(* PLC project shuttle_control, Dassault Systèmes ControlBuild 2024x *)
(* stored: creationDateTime 2023-10-03T11:13:58-01:00 *)

FUNCTION_BLOCK tri_chain.shuttle_control
  VAR_INPUT
    globalRunning : BOOL := false;
    sensorPos1 : BOOL := false;
    sensorPos2 : BOOL := false;
    sensorPos3 : BOOL := false;
    requestCapture1 : BOOL := false;
    endCapture1 : BOOL := false;
    requestCapture2 : BOOL := false;
    endCapture2 : BOOL := false;
    requestCapture3 : BOOL := false;
    endCapture3 : BOOL := false;
    depositRequest : BOOL := false;
    depositFinished : BOOL := false;
  END_VAR
  VAR_OUTPUT
    enableCapture1 : BOOL := false;
    enableCapture2 : BOOL := false;
    enableCapture3 : BOOL := false;
    enableCapture : BOOL := false;
    enableDeposit : BOOL := false;
    moveToLeft : BOOL := false;
    moveToRight : BOOL := false;
  END_VAR
  VAR
    goTo1 : BOOL := false;
    goTo2 : BOOL := false;
    goTo3 : BOOL := false;
    shuttleInPosition : BOOL := false;
  END_VAR

INITIAL_STEP 10:
  COMPUTE_FUNCTION_BLOCKS(S);
END_STEP
TRANSITION FROM 10 TO 11
  := requestCapture1 AND globalRunning;
END_TRANSITION
TRANSITION FROM 10 TO 13
  := requestCapture2 AND globalRunning;
END_TRANSITION
TRANSITION FROM 10 TO 15
  := requestCapture3 AND globalRunning;
END_TRANSITION
INITIAL_STEP 20:
END_STEP
TRANSITION FROM 20 TO 21
  := goTo2 AND NOT sensorPos2;
END_TRANSITION
TRANSITION FROM 20 TO 22
  := goTo2 AND sensorPos2;
END_TRANSITION
INITIAL_STEP 30:
END_STEP
TRANSITION FROM 30 TO 31
  := goTo1 AND NOT sensorPos1;
END_TRANSITION
TRANSITION FROM 30 TO 32
  := goTo1 AND sensorPos1;
END_TRANSITION
INITIAL_STEP 40:
END_STEP
TRANSITION FROM 40 TO 41
  := goTo3 AND NOT sensorPos3;
END_TRANSITION
TRANSITION FROM 40 TO 42
  := goTo3 AND sensorPos3;
END_TRANSITION
STEP 15:
  15_INLINE1(N);
END_STEP
ACTION 15_INLINE1:
  goTo3;
END_ACTION
TRANSITION FROM 15 TO 16
  := shuttleInPosition;
END_TRANSITION
STEP 13:
  13_INLINE2(N);
END_STEP
ACTION 13_INLINE2:
  goTo2;
END_ACTION
TRANSITION FROM 13 TO 14
  := shuttleInPosition;
END_TRANSITION
STEP 11:
  11_INLINE3(N);
END_STEP
ACTION 11_INLINE3:
  goTo1;
END_ACTION
TRANSITION FROM 11 TO 12
  := shuttleInPosition;
END_TRANSITION
STEP 16:
  16_INLINE4(N);
END_STEP
ACTION 16_INLINE4:
  enableCapture;
  enableCapture3;
END_ACTION
TRANSITION FROM 16 TO 17
  := endCapture3 AND depositRequest;
END_TRANSITION
STEP 14:
  14_INLINE5(N);
END_STEP
ACTION 14_INLINE5:
  enableCapture;
  enableCapture2;
END_ACTION
TRANSITION FROM 14 TO 17
  := endCapture2 AND depositRequest;
END_TRANSITION
STEP 12:
  12_INLINE6(N);
END_STEP
ACTION 12_INLINE6:
  enableCapture;
  enableCapture1;
END_ACTION
TRANSITION FROM 12 TO 17
  := endCapture1 AND depositRequest;
END_TRANSITION
STEP 17:
  17_INLINE7(N);
END_STEP
ACTION 17_INLINE7:
  goTo3;
END_ACTION
TRANSITION FROM 17 TO 18
  := shuttleInPosition;
END_TRANSITION
STEP 18:
  18_INLINE8(N);
END_STEP
ACTION 18_INLINE8:
  enableDeposit;
END_ACTION
TRANSITION FROM 18 TO 19
  := depositFinished;
END_TRANSITION
STEP 21:
  21_INLINE9(N);
END_STEP
ACTION 21_INLINE9:
  moveToLeft;
END_ACTION
TRANSITION FROM 21 TO 22
  := sensorPos2;
END_TRANSITION
STEP 19:
  19_INLINE10(N);
END_STEP
ACTION 19_INLINE10:
  goTo2;
END_ACTION
TRANSITION FROM 19 TO 10
  := shuttleInPosition;
END_TRANSITION
STEP 22:
  22_INLINE11(N);
END_STEP
ACTION 22_INLINE11:
  shuttleInPosition;
END_ACTION
TRANSITION FROM 22 TO 20
  := TRUE;
END_TRANSITION
STEP 31:
  31_INLINE12(N);
END_STEP
ACTION 31_INLINE12:
  moveToLeft;
END_ACTION
TRANSITION FROM 31 TO 32
  := sensorPos1;
END_TRANSITION
STEP 41:
  41_INLINE13(N);
END_STEP
ACTION 41_INLINE13:
  moveToRight;
END_ACTION
TRANSITION FROM 41 TO 42
  := sensorPos3;
END_TRANSITION
STEP 32:
  32_INLINE14(N);
END_STEP
ACTION 32_INLINE14:
  shuttleInPosition;
END_ACTION
TRANSITION FROM 32 TO 30
  := TRUE;
END_TRANSITION
STEP 42:
  42_INLINE15(N);
END_STEP
ACTION 42_INLINE15:
  shuttleInPosition;
END_ACTION
TRANSITION FROM 42 TO 40
  := TRUE;
END_TRANSITION
ACTION COMPUTE_FUNCTION_BLOCKS:  (* blocks drawn on the SFC sheet *)
  G1:
  G2:
  G3:
  G4:
END_ACTION
END_FUNCTION_BLOCK
